(* CoDeSys 2.3 export: POINT.EXP *)

(* Data type *)
TYPE POINT :
STRUCT
	X,Y: DINT;
END_STRUCT
END_TYPE
